// TIA Portal V19 export
DATA_BLOCK "Grosse data"   // DB1
   VAR RETAIN
      "Grosse donnée" : Bool;
      "Une autre grosse donnée" : Int;
   END_VAR
BEGIN
END_DATA_BLOCK
